// Mitsubishi GX Works2 project: epeltawer   PLC: FX1N/FX1NC

PROGRAM MAIN
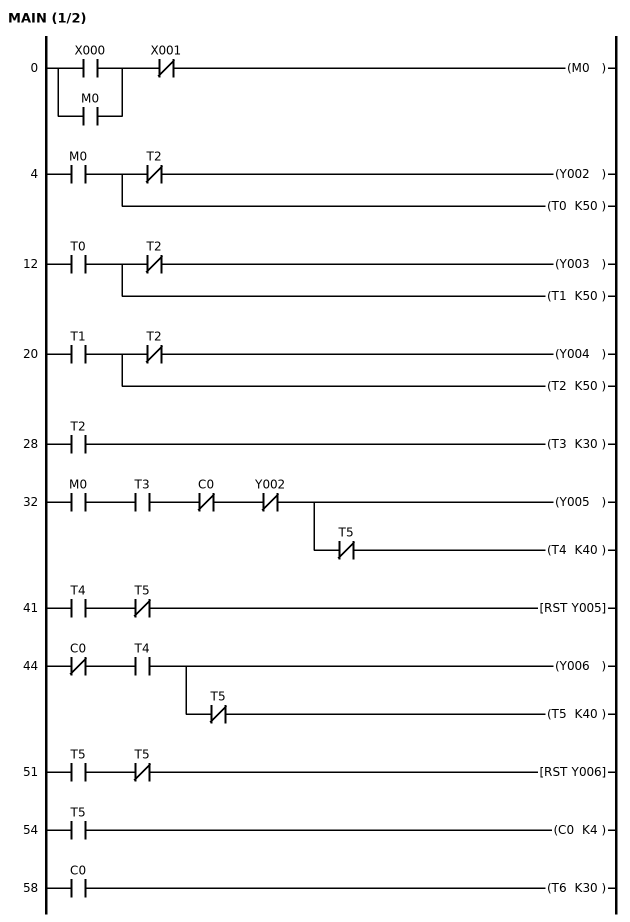
0     LD      X000
      OR      M0
      ANI     X001
      OUT     M0
4     LD      M0
      MPS
      ANI     T2
      OUT     Y002
      MPP
      OUT     T0 K50
12    LD      T0
      MPS
      ANI     T2
      OUT     Y003
      MPP
      OUT     T1 K50
20    LD      T1
      MPS
      ANI     T2
      OUT     Y004
      MPP
      OUT     T2 K50
28    LD      T2
      OUT     T3 K30
32    LD      M0
      AND     T3
      ANI     C0
      ANI     Y002
      OUT     Y005
      ANI     T5
      OUT     T4 K40
41    LD      T4
      ANI     T5
      RST     Y005
44    LDI     C0
      AND     T4
      OUT     Y006
      ANI     T5
      OUT     T5 K40
51    LD      T5
      ANI     T5
      RST     Y006
54    LD      T5
      OUT     C0 K4
58    LD      C0
      OUT     T6 K30
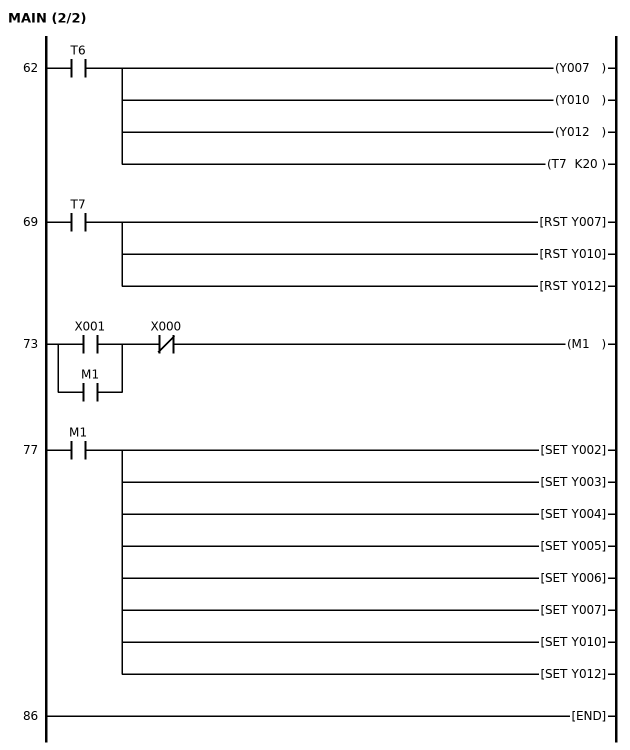
62    LD      T6
      OUT     Y007
      OUT     Y010
      OUT     Y012
      OUT     T7 K20
69    LD      T7
      RST     Y007
      RST     Y010
      RST     Y012
73    LD      X001
      OR      M1
      ANI     X000
      OUT     M1
77    LD      M1
      SET     Y002
      SET     Y003
      SET     Y004
      SET     Y005
      SET     Y006
      SET     Y007
      SET     Y010
      SET     Y012
86    END
END_PROGRAM
